FUNCTION SIGN_I (* this function return true if the integer input is negative *)
  (* Standard: 61499-1 *)
  (* Version 1.0, 2025-12-21, franz *)
  PACKAGE OSCAT::Basic::POUs::Mathematical;
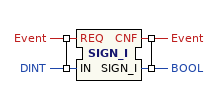
  EVENT_INPUT
    REQ WITH IN;
  END_EVENT
  EVENT_OUTPUT
    CNF WITH SIGN_I;
  END_EVENT
  VAR_INPUT
    IN : DINT;
  END_VAR
  VAR_OUTPUT
    SIGN_I : BOOL;
  END_VAR
  BODY IN ST:
PACKAGE OSCAT::Basic::POUs::Mathematical;

(* this function return true if the integer input is negative *)
FUNCTION SIGN_I : BOOL
VAR_INPUT
	IN : DINT;
END_VAR

(*
 * version 1.3	27. oct. 2008 programmer 	hugo tested by	tobias
 *
 * this function return true if the integer input is negative
 *)
SIGN_I := IN < 0;

END_FUNCTION

(* revision history hm 3.3.2007	rev 1.1 changed method of function for better compatibility to
 * other systems
 *
 * hm	1.12.2007	rev 1.2 changed code to improve performance
 *
 * hm	27. oct. 2008	rev 1.3 changed type of input to dint *)
  END_BODY
END_FUNCTION
